TYPE ST_CSV_Record :
STRUCT
	sName 	: T_MaxString 	:= '';
	nNumber	: UDINT 		:= 0;
	fPos	: LREAL 		:= 0.0;
	bOP		: BOOL 			:= FALSE;
	sDesc	: STRING(40)	:= '';
	data	: ARRAY[0..7] OF BYTE;
END_STRUCT
END_TYPE

(* stored: Version 1.1.0.1, ProductVersion 3.1.4024.12
   DUT ST_CSV_Record: Id {4c50c807-779a-481a-a855-81e148c864e5} *)
